PROGRAM MAIN
VAR
END_VAR

POU();

END_PROGRAM

(* stored: Version 1.1.0.1, ProductVersion 3.1.4024.12
   POU MAIN: Id {01378515-806b-4b83-af62-a943bd4a0113}, SpecialFunc None *)
